// Mitsubishi GX Works2 project: ex   PLC: Q02U

PROGRAM MAIN
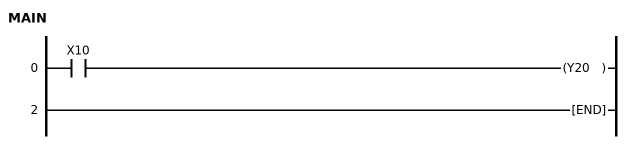
0     LD      X10
      OUT     Y20
2     END
END_PROGRAM
